// VISUs/Templates/GUI_TEMPLATE_USB_COMM
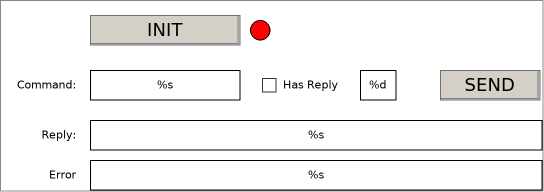
VISUALIZATION GUI_TEMPLATE_USB_COMM  // 544x192
VAR_IN_OUT
	m_Instance:	FB_ADS_COMM;
END_VAR
VAR
	cmd:			STRING;
	bHasReply:		BOOL;		(* If TRUE, there is a reply to the command *)
	nNumReplies:	DINT;	(* Number of replies, i.e. number of cfg.sReplySuffix strings expected in the reply *)
END_VAR
    Button (440,70 100x30), "SEND"
        OnMouseClick: execute {
            m_Instance.ctrl.nCommand:=2;
            m_Instance.ctrl.sCmd:=cmd;
            m_Instance.ctrl.bHasReply:=bHasReply;
            m_Instance.ctrl.nNumReplies:=nNumReplies;
            m_Instance.ctrl.bExecute:=TRUE;
        }
    Rectangle (90,120 452x30), "%s", text variable: m_Instance.stat.sReply
    Rectangle (90,70 150x30), "%s", tooltip "Command (without terminators)", text variable: cmd
        OnMouseClick: write the text variable via Default
    Button (90,15 150x30), "INIT", tooltip "Initialize communication"
        OnMouseClick: execute { m_Instance.ctrl.nCommand:=1; m_Instance.ctrl.bExecute:=TRUE; }
    Checkbox (260,70 97x30), "Has Reply", tooltip "Check this box if reply is expected", variable: bHasReply
    Rectangle (360,70 36x30), "%d", tooltip "Set the number of expected replies", text variable: nNumReplies, input disabled if: FALSE
        OnMouseClick: write the text variable via Default, min 0
    Label (10,70 69x30), "Command:"
    Label (10,120 69x30), "Reply:"
    Label (10,160 69x30), "Error"
    Rectangle (90,160 452x30), "%s", text variable: m_Instance.stat.sErrorText
    Ellipse (250,20 20x20), tooltip "GREEN=Initialized RED=Not-initialized", text variable: m_Instance.stat.bInitialised, colour toggle: m_Instance.stat.bInitialised
END_VISUALIZATION

// VISUs/GUI_ADS_COMM_TEST
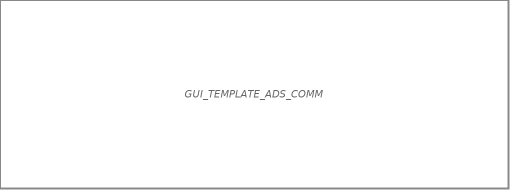
VISUALIZATION GUI_ADS_COMM_TEST  // 510x190
    Frame (0,0 508x188)
        shows GUI_TEMPLATE_ADS_COMM(m_Instance := MAIN.USB1)
END_VISUALIZATION

// VISUs/GUI_CCC
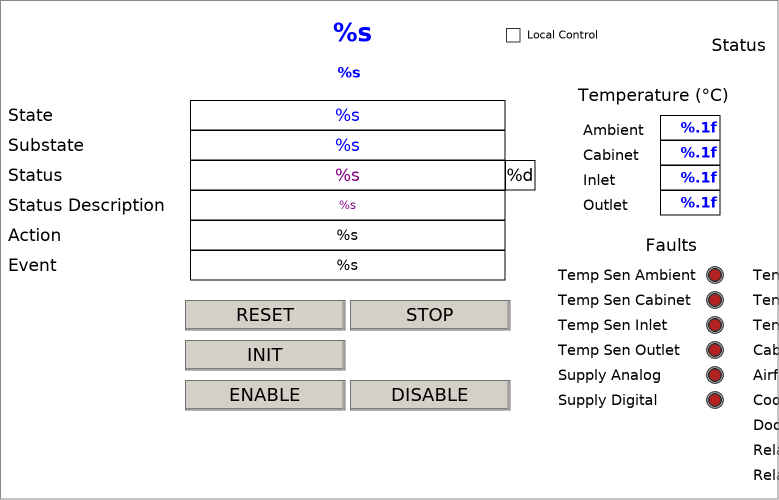
VISUALIZATION GUI_CCC  // 779x500
    Frame (0,0 777x498)
        shows GUI_TEMPLATE_CCC(m_Instance := MAIN.CCC)
END_VISUALIZATION

// VISUs/GUI_LAKESHORE_340
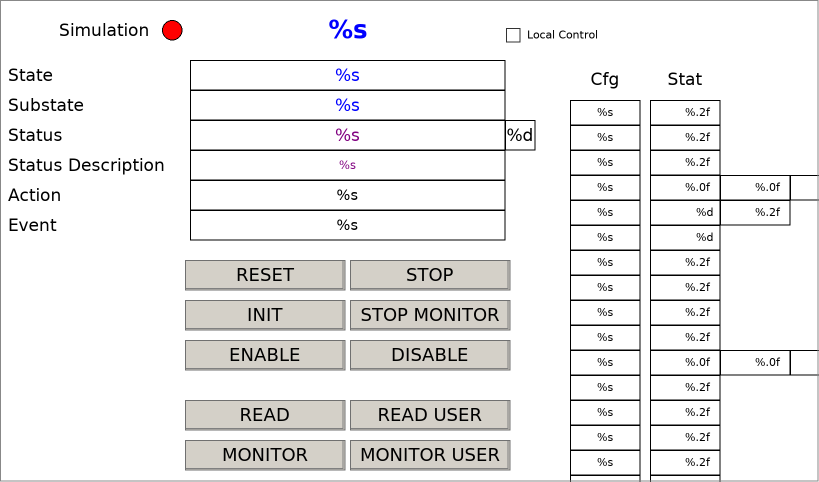
VISUALIZATION GUI_LAKESHORE_340  // 819x482
    Frame (0,0 817x480)
        shows GUI_TEMPLATE_LAKESHORE_340(m_Instance := MAIN.LS340)
END_VISUALIZATION
